{attribute 'linkalways'} 
{attribute 'no_explicit_call' := 'This FB is a CLASS and must be accessed using methods or properties'}
{attribute 'enable_dynamic_creation'}
FUNCTION_BLOCK Node_F_VN_AddToContainerElements_TcVnVector2_USINT EXTENDS VisionNode
VAR
    aValue : _TcVnVector2_USINT;
    ipContainer : _ITcVnContainer;
    hrPrev : _HRESULT(S_OK);
    hresult : _HRESULT(S_OK);
END_VAR

METHOD PUBLIC  Clone : I_Node
VAR
    pNode : POINTER TO Node_F_VN_AddToContainerElements_TcVnVector2_USINT;
END_VAR
pNode := __NEW(Node_F_VN_AddToContainerElements_TcVnVector2_USINT);
Clone := pNode^;
END_METHOD

METHOD FB_init : BOOL
VAR_INPUT
    bInitRetains : BOOL; // if TRUE, the retain variables are initialized (warm start / cold start)
    bInCopyCode : BOOL;  // if TRUE, the instance afterwards gets moved into the copy code (online change)
END_VAR
AddInput('aValue', aValue);
AddInput('ipContainer', ipContainer);
AddInput('hrPrev', hrPrev);
AddOutput('ipContainer', ipContainer);
AddOutput('hresult',hresult);
END_METHOD

METHOD PROTECTED OnExecute : HRESULT
hresult.Value := F_VN_AddToContainerElements_TcVnVector2_USINT(
    aValue := aValue.Value,
    ipContainer := ipContainer.Value,
    hrPrev:= hrPrev.Value);
END_METHOD

METHOD PUBLIC PreExecutionCheck
VAR_INPUT
    Check : I_PreExecutionChecks;
END_VAR
Check.IsTrue(ipContainer.IsValid, 'ipContainer must be a valid container');
Check.IsTrue(ipContainer.HasType(TC_GLOBAL_CONST_LIST.ContainerType_Vector_TcVnVector2_USINT), 'ipContainer contains incorrect type');
END_METHOD

END_FUNCTION_BLOCK

(* stored: Version 1.1.0.1, ProductVersion 3.1.4024.13
   POU Node_F_VN_AddToContainerElements_TcVnVector2_USINT: Id {67892d0f-3ab0-46df-a83c-7ac37595fc0d}, SpecialFunc None
   Folder Constructor: Id {7b738df7-68ac-4a53-b88e-2b9700eb15ea}
   Method Clone: Id {c418c7ef-756d-4f58-ac5f-ecfc4945c526}
   Method FB_init: Id {efa7ebe6-226a-4119-8512-2b30a41c31f4}
   Method OnExecute: Id {8a671a12-ca36-46b5-8f08-d8282a4ba02f}
   Method PreExecutionCheck: Id {d2d156e3-2a62-4ded-bdea-3c8709391312} *)
